ABB RobotStudio station: EstacionLabsirIRB2.rsstn

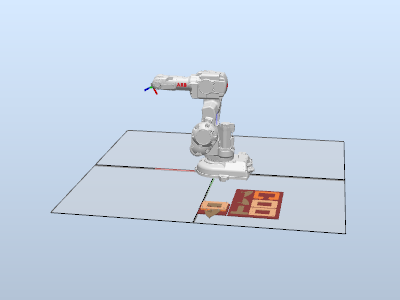
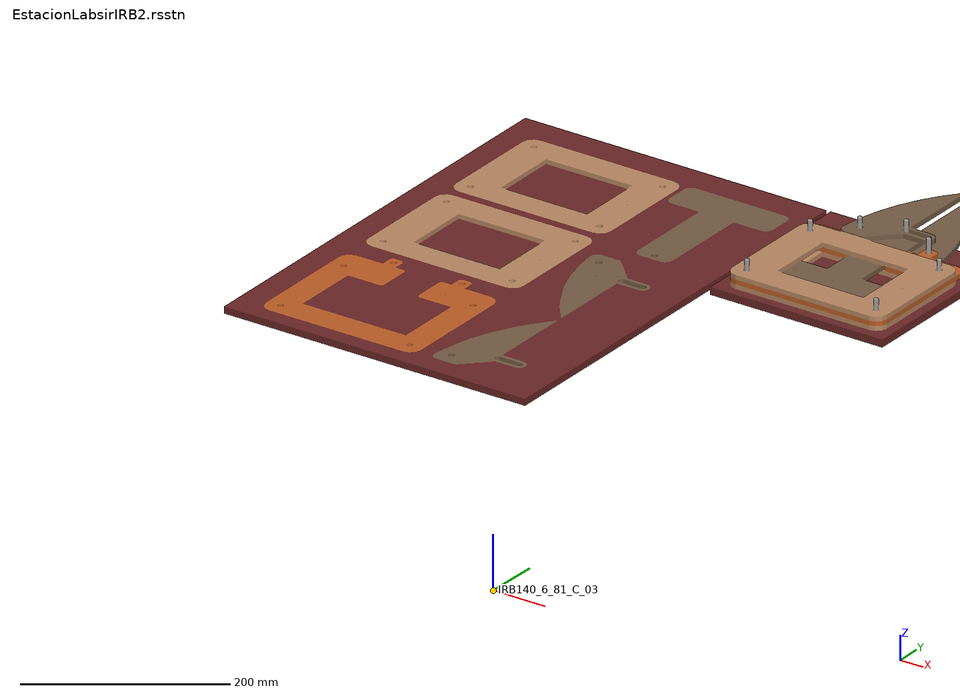
[picture v1: parts stored in the station drawn from their meshes, with robot base, taught points and paths (robot models come from the ABB library and are not in the file)]
Station Station (saved by RobotStudio 22.2.9947.0)
Controller IRB140_6_81
  mechanical unit ROB_1: IRB140_6_81_C_03, 6 joints, base frame (0, 0, 0) mm
Layout (positions relative to the parent item):
  - IRB140_6_81_C_03 [mechanism, from Robots\IRB140_6_81_C_G_03.rslib] at (0, 0, 0) mm; joint values [0, 0, 0, 0, 0.5237, 0] (rad or m)
  - PortaPiezas [part] at (-375, 600, 0) mm, rotated rx 0 ry 0 rz 90 deg, size 500 x 350 x 7 mm
  - BaseEnsamble [part] at (-100, 750, 0) mm, rotated rx 0 ry 0 rz 90 deg, size 282.5 x 200 x 35 mm
